INTERFACE I_AdsAddr

{attribute 'monitoring':='call'}
PROPERTY NetId : T_AmsNetID
GET
END_GET
END_PROPERTY

{attribute 'monitoring':='call'}
PROPERTY Port : WORD
GET
END_GET
END_PROPERTY

END_INTERFACE

(* stored: Version 1.1.0.1, ProductVersion 3.1.4024.12
   Itf I_AdsAddr: Id {18279f44-fbe6-4ebb-8976-868ddae2bc22}
   Property NetId: Id {e8ac5ac4-0807-4420-a1ca-07ef4666c853}
   Get Get: Id {9781502f-5cfc-4463-938e-9980bd1c58ef}
   Property Port: Id {fcde7741-8a7f-4078-acba-893ed034d6cb}
   Get Get: Id {b1a17193-afa5-4eab-a1d1-28dfbf5adb0d} *)
